// Mitsubishi GX Works2 project: plc_group_21   PLC: FX3G

// global labels: Global1
VAR_GLOBAL
  input_switch AT M10 : BOOL;
  clementine_input AT D1200 : REAL;
  orange_input AT D1202 : REAL;
  pomela_input AT D1204 : REAL;
  clementine_container AT D1100 : REAL;
  orange_container AT D1102 : REAL;
  pomela_container AT D1104 : REAL;
  start_day_switch AT X010 : BOOL;
  input_ratio AT D1106 : REAL;
  start_day_light AT Y010 : BOOL;
  input_ratio_OC AT D1106 : REAL;
  input_ratio_PO AT D1108 : REAL;
  start_day_success AT M11 : BOOL;
  start_wash AT X002 : BOOL;
  wash_timer AT TC0 : BOOL;
  wash_is_on_light AT Y005 : BOOL;
END_VAR
VAR_GLOBAL CONSTANT
  const2 : REAL := 2.0;
END_VAR
VAR_GLOBAL
  const_ratio_input AT D1212 : REAL;
  const_ratio AT D1112 : REAL;
  recipe AT D1114 : REAL;
  recipe_input AT D1214 : REAL;
  orange_container_stock AT D1126 : REAL;
  recipe_2 AT D1116 : REAL;
  clementine_container_stock AT D1118 : REAL;
  pomela_container_stock AT D1120 : REAL;
  finish_wash_light AT M12 : BOOL;
  start_collecting AT X001 : BOOL;
  start_collecting_light AT Y001 : BOOL;
  stop_collecting_light AT M13 : BOOL;
  add_to_collecting AT M14 : BOOL;
  add_to_collecting_light AT M14 : BOOL;
  all_fruits_for_squeezing AT D1122 : REAL;
  ready_for_squeezing_light AT M15 : BOOL;
  start_squeezing_switch AT X011 : BOOL;
  start_squeez_counter AT CC0 : BOOL;
END_VAR
VAR_GLOBAL CONSTANT
  button_counter : INT := 2;
END_VAR
VAR_GLOBAL
  start_squeez_counter_cs AT CS0 : BOOL;
  wash_timer_ts AT TS0 : BOOL;
END_VAR
VAR_GLOBAL CONSTANT
  squeezing_timer : INT := 1;
END_VAR
VAR_GLOBAL
  start_squeezing_ts AT TS1 : BOOL;
  sqeezing_light_2 AT Y002 : BOOL;
  squeezing_light_3 AT Y003 : BOOL;
  squeez_help AT M16 : BOOL;
  squeez_light_2 AT Y002 : BOOL;
  start_squeezing_1 AT TC1 : BOOL;
  start_squeezing_2 AT TC2 : BOOL;
  start_squeezing_ts2 AT TS2 : BOOL;
  start_squeezing_ts1 AT TS1 : BOOL;
  squeez_light_3 AT Y003 : BOOL;
  end_squeezing AT M17 : BOOL;
  juice_container AT D1124 : REAL;
  squeez_counter AT CS0 : BOOL;
  start_squeezing_timer AT TC3 : BOOL;
END_VAR
VAR_GLOBAL CONSTANT
  squeezing_timer_3s : INT := 30;
  button_counter_2k : INT := 2;
  squeezing_timer_1 : INT := 10;
END_VAR
VAR_GLOBAL
  start_squeez_counter_ts AT TS3 : BOOL;
  stop_squeez_timer AT M13 : BOOL;
  ready_for_quality AT M18 : BOOL;
  quality_switch AT X003 : BOOL;
  analog_input_2 AT D8281 : INT;
  quality_input_real AT D1128 : REAL;
END_VAR
VAR_GLOBAL CONSTANT
  const5 : REAL := 2000;
  const1 : REAL := 400;
END_VAR
VAR_GLOBAL
  quality_success AT M19 : BOOL;
  quality_success_light AT Y004 : BOOL;
  quality_success_stop_light AT TS4 : BOOL;
  start_quality_move AT TC4 : BOOL;
END_VAR
VAR_GLOBAL CONSTANT
  quality_move_timer_5s : INT := 50;
END_VAR
VAR_GLOBAL
  start_quality_move_ts AT TS4 : BOOL;
  juice_storage AT D1132 : REAL;
  ready_juice AT M20 : BOOL;
  start_quality_count AT CC1 : BOOL;
END_VAR
VAR_GLOBAL CONSTANT
  quality_counter_2k : INT := 2;
END_VAR
VAR_GLOBAL
  quality_count AT CS1 : BOOL;
END_VAR
VAR_GLOBAL CONSTANT
  const0 : REAL;
END_VAR
VAR_GLOBAL
  daily_juice_count AT D1130 : REAL;
  stop_work AT X007 : BOOL;
  check_daily_count AT X004 : BOOL;
  analog_output AT D8282 : REAL;
  check_daily_count_light AT Y011 : BOOL;
  reset_iteration AT M22 : BOOL;
  reset_day AT M23 : BOOL;
  reset_break AT M23 : BOOL;
END_VAR
VAR_GLOBAL CONSTANT
  const_3s : INT := 30;
END_VAR
VAR_GLOBAL
  reset_all AT X007 : BOOL;
  reset_all_timer AT TC7 : BOOL;
END_VAR
VAR_GLOBAL CONSTANT
  reset_all_timer_3s : INT := 30;
END_VAR
VAR_GLOBAL
  reset_all_timer_ts AT TS7 : BOOL;
  reset_all_timer_1 AT TC8 : BOOL;
  reset_help AT M70 : BOOL;
  reset_all_timer_2 AT TC9 : BOOL;
  reset_all_timer_1_ts AT TS8 : BOOL;
  reset_all_timer_2_ts AT TS9 : BOOL;
  finish_day AT M80 : BOOL;
  help_close_M12 AT M81 : BOOL;
END_VAR
VAR_GLOBAL CONSTANT
  ready_juice_count : REAL := 1;
  reset_timer_1 : INT := 10;
END_VAR
VAR_GLOBAL
  finish_day_1 AT M85 : BOOL;
  help_count_light AT M86 : BOOL;
END_VAR

// task Task_01 (event TRUE, interval 0, priority 31): POU_01

PROGRAM POU_01
(* structured ladder/FBD written out as ST: instructions are called as NAME(EN, inputs, outputs); _pN, _eN, _tN stand for wires *)
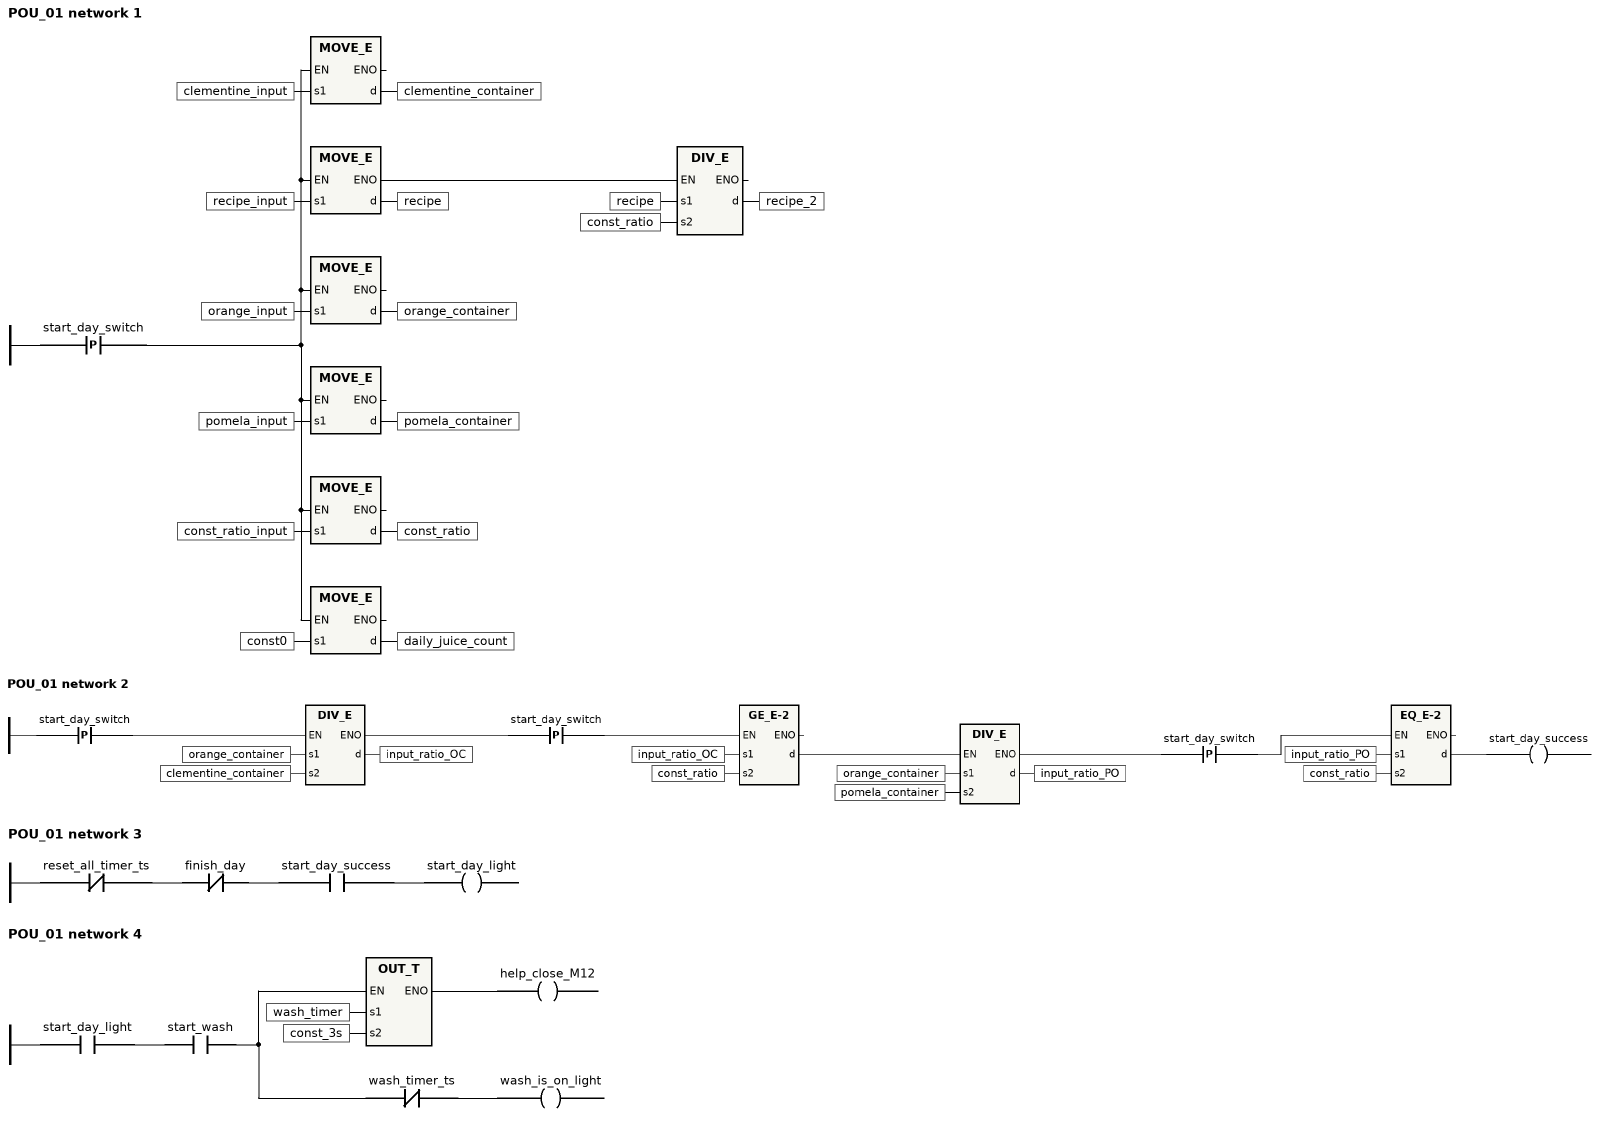
(* network 1 *)
_p1 := LDP(TRUE, start_day_switch);
MOVE_E(_p1, clementine_input, clementine_container);
MOVE_E(_p1, orange_input, orange_container);
MOVE_E(_p1, pomela_input, pomela_container);
MOVE_E(_p1, const_ratio_input, const_ratio);
_e2 := MOVE_E(_p1, recipe_input, recipe);
DIV_E(_e2, recipe, const_ratio, recipe_2);
MOVE_E(_p1, const0, daily_juice_count);
(* network 2 *)
_e1 := DIV_E(LDP(TRUE, start_day_switch), orange_container, clementine_container, input_ratio_OC);
GE_E(_e1 AND LDP(TRUE, start_day_switch), input_ratio_OC, const_ratio, _t2);
_e3 := DIV_E(_t2, orange_container, pomela_container, input_ratio_PO);
EQ_E(_e3 AND LDP(TRUE, start_day_switch), input_ratio_PO, const_ratio, _t4);
start_day_success := _t4;
(* network 3 *)
start_day_light := NOT reset_all_timer_ts AND NOT finish_day AND start_day_success;
(* network 4 *)
_p1 := start_day_light AND start_wash;
_e2 := OUT_T(_p1, wash_timer, const_3s);
help_close_M12 := _e2;
wash_is_on_light := _p1 AND NOT wash_timer_ts;
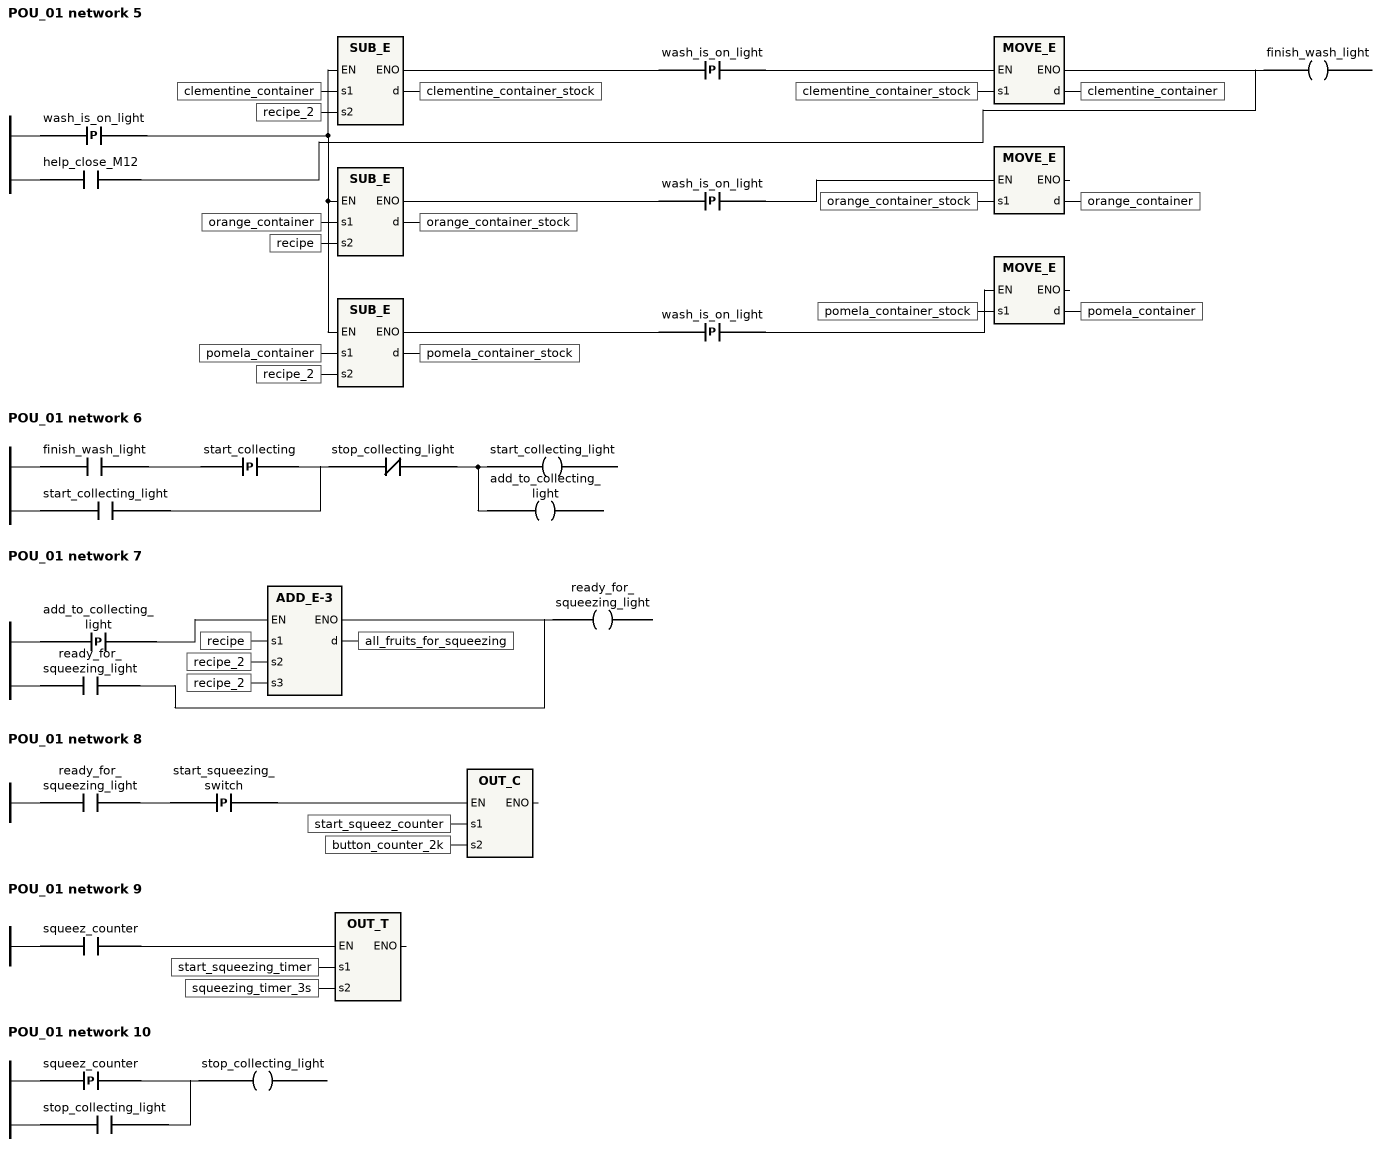
(* network 5 *)
_p1 := LDP(TRUE, wash_is_on_light);
_e2 := SUB_E(_p1, orange_container, recipe, orange_container_stock);
MOVE_E(_e2 AND LDP(TRUE, wash_is_on_light), orange_container_stock, orange_container);
_e3 := SUB_E(_p1, clementine_container, recipe_2, clementine_container_stock);
_e4 := MOVE_E(_e3 AND LDP(TRUE, wash_is_on_light), clementine_container_stock, clementine_container);
finish_wash_light := _e4 OR help_close_M12;
_e5 := SUB_E(_p1, pomela_container, recipe_2, pomela_container_stock);
MOVE_E(_e5 AND LDP(TRUE, wash_is_on_light), pomela_container_stock, pomela_container);
(* network 6 *)
_p1 := ((finish_wash_light AND LDP(TRUE, start_collecting)) OR start_collecting_light) AND NOT stop_collecting_light;
start_collecting_light := _p1;
add_to_collecting_light := _p1;
(* network 7 *)
_e1 := ADD_E(LDP(TRUE, add_to_collecting_light), recipe, recipe_2, recipe_2, all_fruits_for_squeezing);
ready_for_squeezing_light := _e1 OR ready_for_squeezing_light;
(* network 8 *)
OUT_C(ready_for_squeezing_light AND LDP(TRUE, start_squeezing_switch), start_squeez_counter, button_counter_2k);
(* network 9 *)
OUT_T(squeez_counter, start_squeezing_timer, squeezing_timer_3s);
(* network 10 *)
stop_collecting_light := LDP(TRUE, squeez_counter) OR stop_collecting_light;
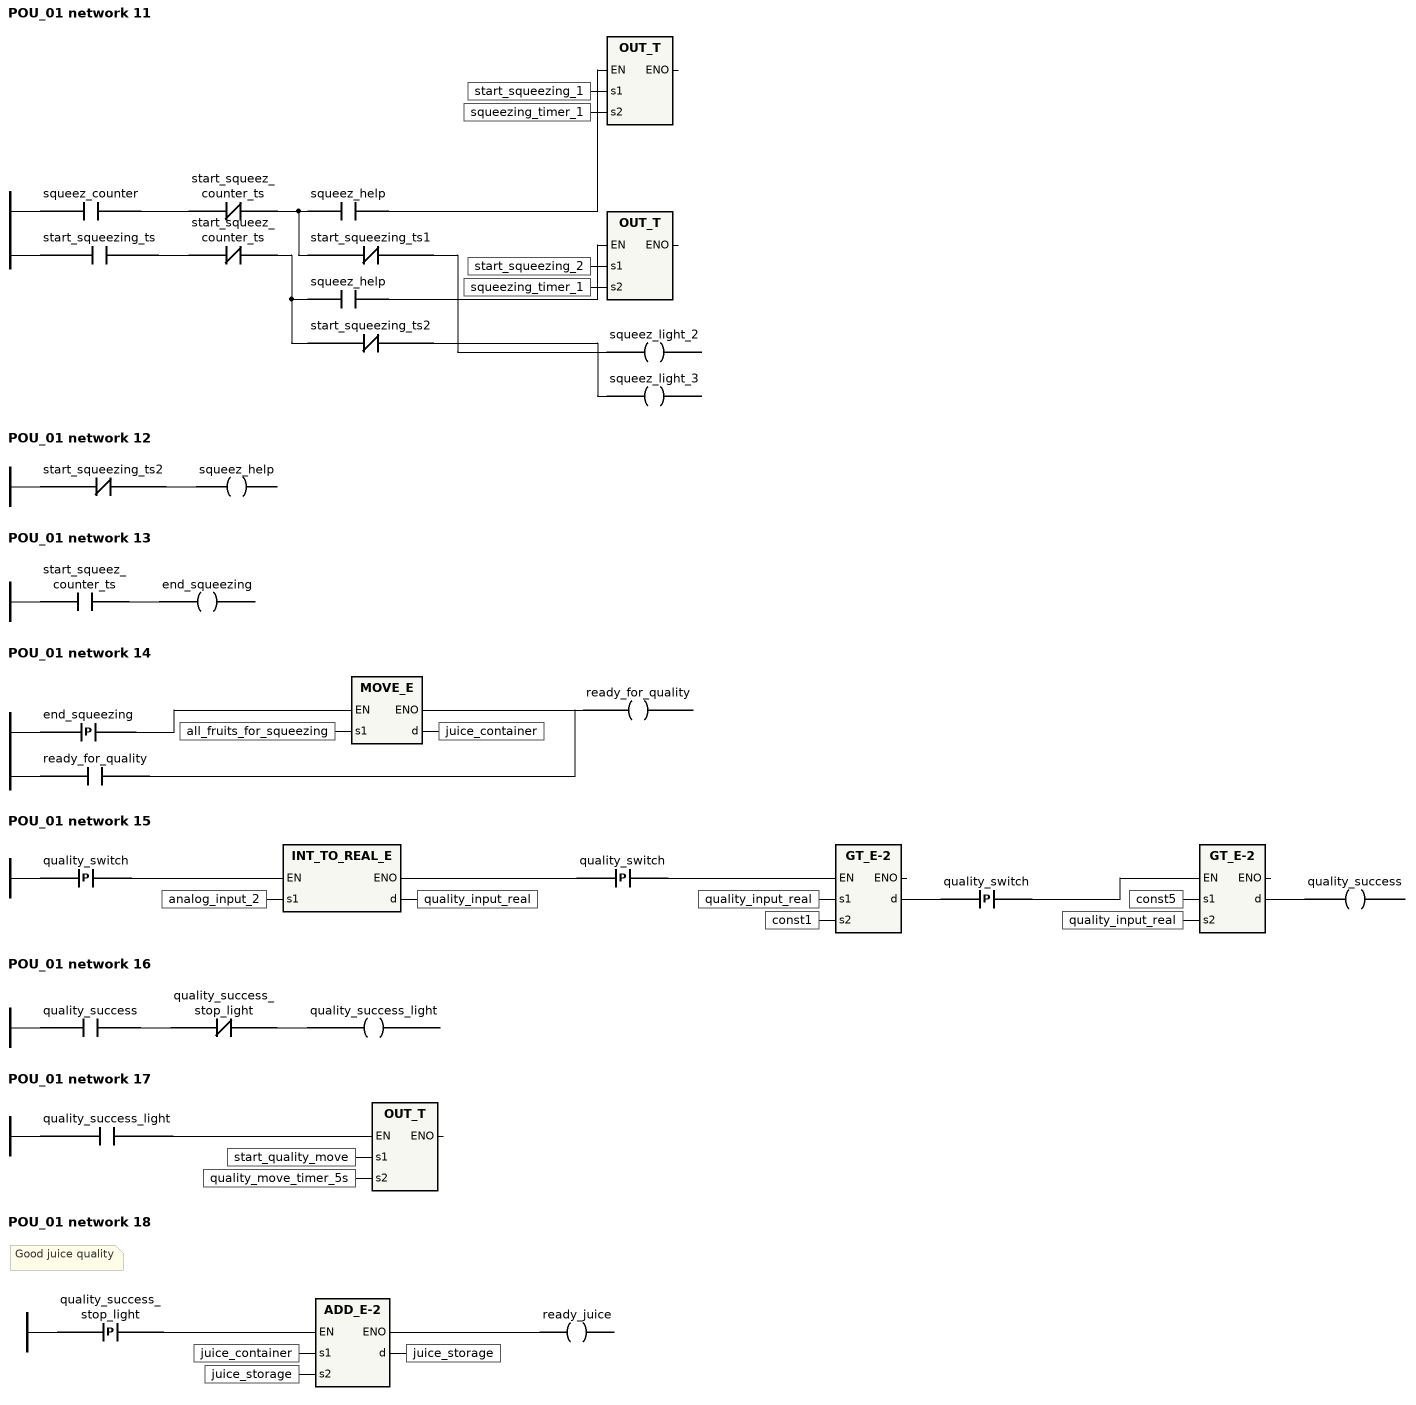
(* network 11 *)
_p1 := squeez_counter AND NOT start_squeez_counter_ts;
OUT_T(_p1 AND squeez_help, start_squeezing_1, squeezing_timer_1);
squeez_light_2 := _p1 AND NOT start_squeezing_ts1;
_p2 := start_squeezing_ts AND NOT start_squeez_counter_ts;
OUT_T(_p2 AND squeez_help, start_squeezing_2, squeezing_timer_1);
squeez_light_3 := _p2 AND NOT start_squeezing_ts2;
(* network 12 *)
squeez_help := NOT start_squeezing_ts2;
(* network 13 *)
end_squeezing := start_squeez_counter_ts;
(* network 14 *)
_e1 := MOVE_E(LDP(TRUE, end_squeezing), all_fruits_for_squeezing, juice_container);
ready_for_quality := _e1 OR ready_for_quality;
(* network 15 *)
_e1 := INT_TO_REAL_E(LDP(TRUE, quality_switch), analog_input_2, quality_input_real);
GT_E(_e1 AND LDP(TRUE, quality_switch), quality_input_real, const1, _t2);
GT_E(_t2 AND LDP(TRUE, quality_switch), const5, quality_input_real, _t3);
quality_success := _t3;
(* network 16 *)
quality_success_light := quality_success AND NOT quality_success_stop_light;
(* network 17 *)
OUT_T(quality_success_light, start_quality_move, quality_move_timer_5s);
(* network 18 *)
(* Good juice quality *)
_e1 := ADD_E(LDP(TRUE, quality_success_stop_light), juice_container, juice_storage, juice_storage);
ready_juice := _e1;
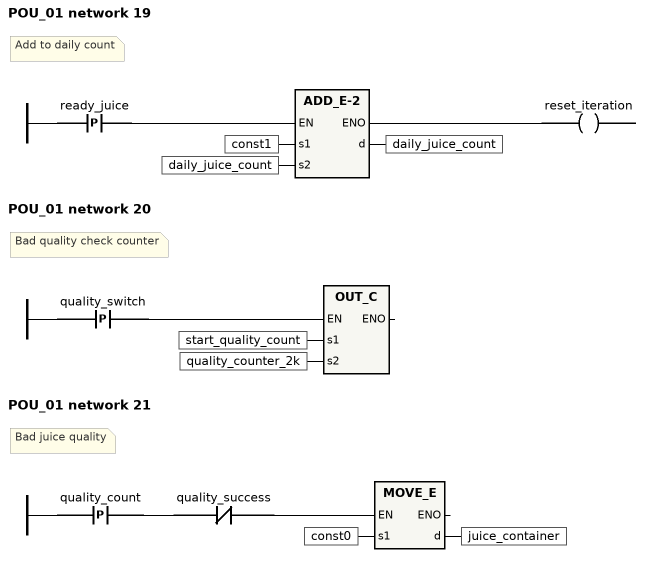
(* network 19 *)
(* Add to daily count *)
_e1 := ADD_E(LDP(TRUE, ready_juice), const1, daily_juice_count, daily_juice_count);
reset_iteration := _e1;
(* network 20 *)
(* Bad quality check counter *)
OUT_C(LDP(TRUE, quality_switch), start_quality_count, quality_counter_2k);
(* network 21 *)
(* Bad juice quality *)
MOVE_E(LDP(TRUE, quality_count) AND NOT quality_success, const0, juice_container);
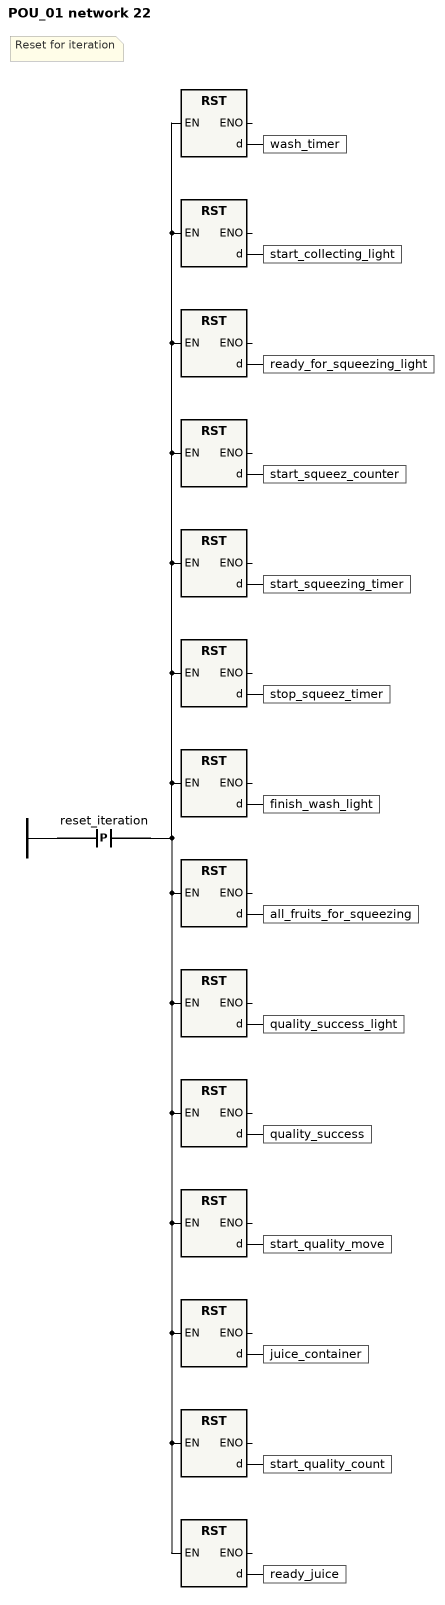
(* network 22 *)
(* Reset for iteration *)
_p1 := LDP(TRUE, reset_iteration);
RST(_p1, wash_timer);
RST(_p1, start_collecting_light);
RST(_p1, ready_for_squeezing_light);
RST(_p1, start_squeez_counter);
RST(_p1, start_squeezing_timer);
RST(_p1, stop_squeez_timer);
RST(_p1, finish_wash_light);
RST(_p1, all_fruits_for_squeezing);
RST(_p1, quality_success_light);
RST(_p1, quality_success);
RST(_p1, start_quality_move);
RST(_p1, juice_container);
RST(_p1, start_quality_count);
RST(_p1, ready_juice);
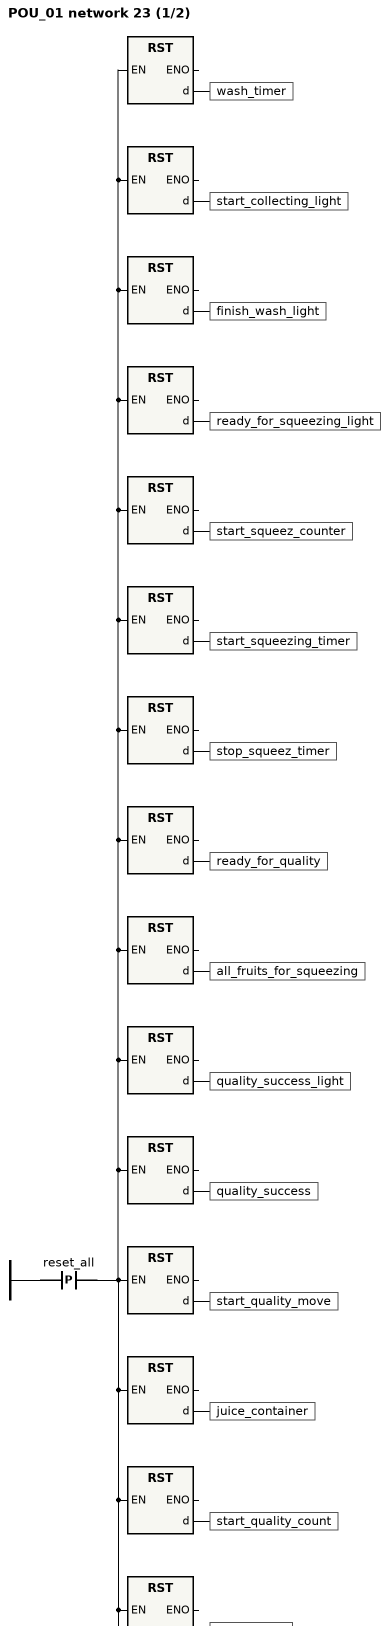
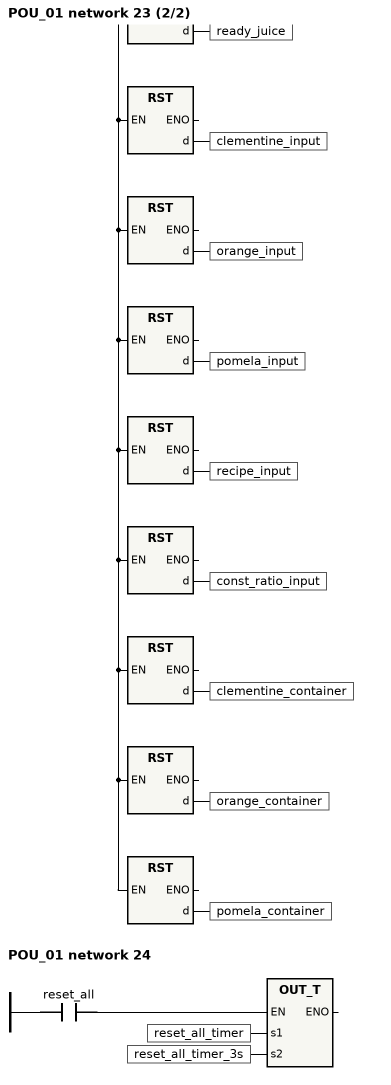
(* network 23 *)
_p1 := LDP(TRUE, reset_all);
RST(_p1, wash_timer);
RST(_p1, start_collecting_light);
RST(_p1, finish_wash_light);
RST(_p1, ready_for_squeezing_light);
RST(_p1, start_squeez_counter);
RST(_p1, start_squeezing_timer);
RST(_p1, stop_squeez_timer);
RST(_p1, ready_for_quality);
RST(_p1, all_fruits_for_squeezing);
RST(_p1, quality_success_light);
RST(_p1, quality_success);
RST(_p1, start_quality_move);
RST(_p1, juice_container);
RST(_p1, start_quality_count);
RST(_p1, ready_juice);
RST(_p1, clementine_input);
RST(_p1, orange_input);
RST(_p1, pomela_input);
RST(_p1, recipe_input);
RST(_p1, const_ratio_input);
RST(_p1, clementine_container);
RST(_p1, orange_container);
RST(_p1, pomela_container);
(* network 24 *)
OUT_T(reset_all, reset_all_timer, reset_all_timer_3s);
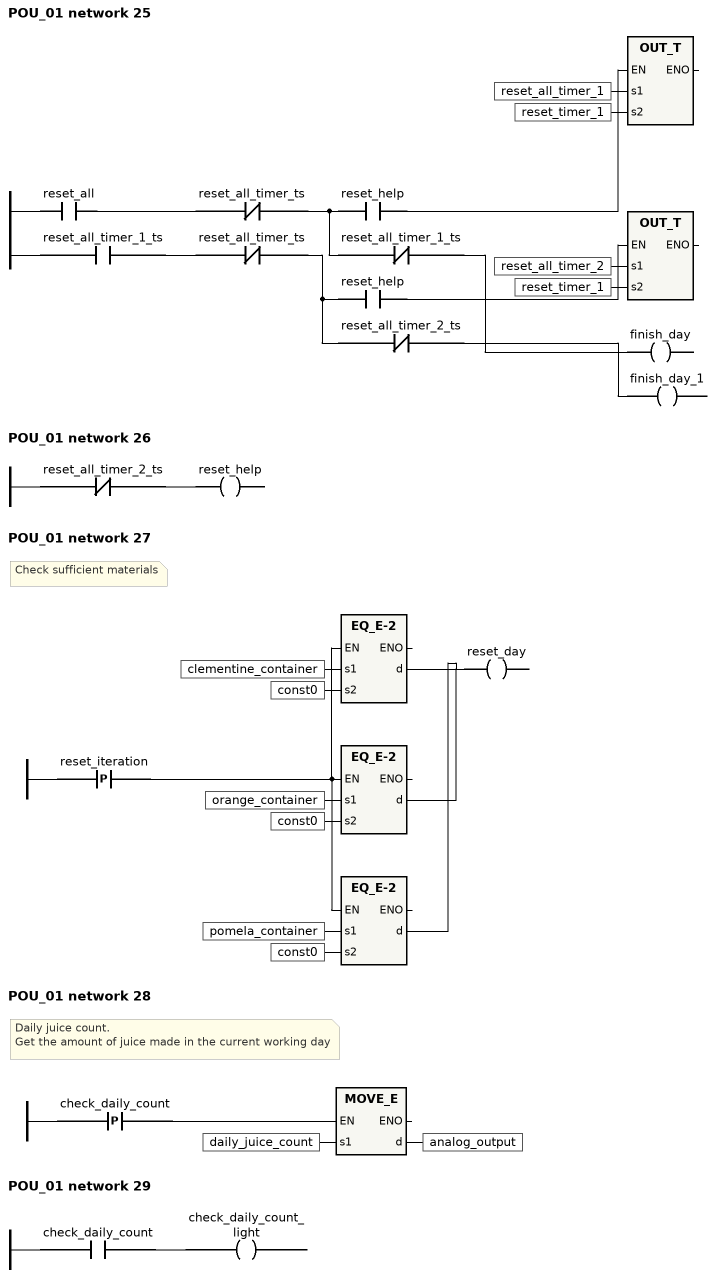
(* network 25 *)
_p1 := reset_all AND NOT reset_all_timer_ts;
OUT_T(_p1 AND reset_help, reset_all_timer_1, reset_timer_1);
finish_day := _p1 AND NOT reset_all_timer_1_ts;
_p2 := reset_all_timer_1_ts AND NOT reset_all_timer_ts;
OUT_T(_p2 AND reset_help, reset_all_timer_2, reset_timer_1);
finish_day_1 := _p2 AND NOT reset_all_timer_2_ts;
(* network 26 *)
reset_help := NOT reset_all_timer_2_ts;
(* network 27 *)
(* Check sufficient materials *)
_p1 := LDP(TRUE, reset_iteration);
EQ_E(_p1, clementine_container, const0, _t2);
EQ_E(_p1, orange_container, const0, _t3);
EQ_E(_p1, pomela_container, const0, _t4);
reset_day := _t2 OR _t3 OR _t4;
(* network 28 *)
(* Daily juice count. / Get the amount of juice made in the current working day *)
MOVE_E(LDP(TRUE, check_daily_count), daily_juice_count, analog_output);
(* network 29 *)
check_daily_count_light := check_daily_count;
END_PROGRAM
